SFTON3D P021
SMOVL C00538 BC00538 V=100.0  +MOVJ EC00538
SFTOF3D
MOVL C00539 BC00539 V=400.0  +MOVJ EC00539 VJ=100.00
SFTON3D P021
SMOVL C00540 BC00540 V=166.7 PL=0  +MOVJ EC00540
SREFP 1 C00541 BC00541  +REFP EC00541
SREFP 2 C00542 BC00542  +REFP EC00542
MACRO1 MJ#(0) ARGF9
ARCON
SMOVL C00543 BC00543 V=12.5  +MOVJ EC00543
SMOVL C00544 BC00544 V=12.5  +MOVJ EC00544
ARCOF
SFTOF3D
MOVL C00545 BC00545 V=400.0  +MOVJ EC00545 VJ=100.00
MOVL C00546 BC00546 V=1000.0  +MOVJ EC00546 VJ=100.00
MOVJ C00547 BC00547 VJ=100.00  +MOVJ EC00547 VJ=100.00
MOVJ C00548 BC00548 VJ=100.00  +MOVJ EC00548 VJ=100.00
MOVJ C00549 BC00549 VJ=100.00  +MOVJ EC00549 VJ=100.00
'2
'Path W3693
SFTOF3D
MOVJ C00550 BC00550 VJ=100.00  +MOVJ EC00550 VJ=100.00
MACRO1 MJ#(0) ARGF6
SFTON3D P060
SMOVL C00551 BC00551 V=166.7  +MOVJ EC00551
ARCON
SMOVL C00552 BC00552 V=8.3  +MOVJ EC00552
SMOVL C00553 BC00553 V=8.3  +MOVJ EC00553
SMOVL C00554 BC00554 V=8.3  +MOVJ EC00554
ARCOF
SMOVL C00555 BC00555 V=166.7  +MOVJ EC00555
SMOVL C00556 BC00556 V=333.3  +MOVJ EC00556
MACRO1 MJ#(0) ARGF14
SFTON3D P061
SMOVL C00557 BC00557 V=166.7  +MOVJ EC00557
ARCON
SMOVL C00558 BC00558 V=10.0  +MOVJ EC00558
ARCOF
SFTOF3D
SMOVL C00559 BC00559 V=416.7  +MOVJ EC00559
MOVJ C00560 BC00560 VJ=100.00  +MOVJ EC00560 VJ=25.00
MOVL C00561 BC00561 V=400.0  +MOVJ EC00561 VJ=100.00
SFTON3D P023
SMOVL C00562 BC00562 V=166.7 PL=0  +MOVJ EC00562
SREFP 1 C00563 BC00563  +REFP EC00563
SREFP 2 C00564 BC00564  +REFP EC00564
MACRO1 MJ#(0) ARGF9
ARCON
SMOVL C00565 BC00565 V=11.7  +MOVJ EC00565
ARCOF
SFTOF3D
MOVL C00566 BC00566 V=400.0  +MOVJ EC00566 VJ=100.00
MOVL C00567 BC00567 V=1000.0  +MOVJ EC00567 VJ=100.00
'Path W3694
SFTOF3D
MOVJ C00568 BC00568 VJ=20.00  +MOVJ EC00568 VJ=0.78
MOVJ C00569 BC00569 VJ=100.00  +MOVJ EC00569 VJ=100.00
MOVL C00570 BC00570 V=400.0  +MOVJ EC00570 VJ=100.00
SFTON3D P023
SMOVL C00571 BC00571 V=166.7 PL=0  +MOVJ EC00571
SREFP 1 C00572 BC00572  +REFP EC00572
SREFP 2 C00573 BC00573  +REFP EC00573
ARCON
SMOVL C00574 BC00574 V=11.7  +MOVJ EC00574
ARCOF
SFTOF3D
MOVL C00575 BC00575 V=400.0  +MOVJ EC00575 VJ=100.00
MOVL C00576 BC00576 V=1000.0  +MOVJ EC00576 VJ=100.00
MOVJ C00577 BC00577 VJ=100.00  +MOVJ EC00577 VJ=100.00
MOVJ C00578 BC00578 VJ=100.00  +MOVJ EC00578 VJ=100.00
MOVJ C00579 BC00579 VJ=100.00  +MOVJ EC00579 VJ=100.00
MOVJ C00580 BC00580 VJ=100.00  +MOVJ EC00580 VJ=100.00
SFTOF3D
MOVJ C00581 BC00581 VJ=100.00  +MOVJ EC00581 VJ=100.00
SFTOF3D
MOVJ C00582 BC00582 VJ=100.00  +MOVJ EC00582 VJ=100.00
MOVL C00583 BC00583 V=666.7  +MOVJ EC00583 VJ=100.00
SFTON3D P021
MACRO1 MJ#(0) ARGF9
SMOVL C00584 BC00584 V=166.7 PL=0  +MOVJ EC00584
SREFP 1 C00585 BC00585  +REFP EC00585
SREFP 2 C00586 BC00586  +REFP EC00586
ARCON
SMOVL C00587 BC00587 V=11.7  +MOVJ EC00587
ARCOF
SFTOF3D
MOVL C00588 BC00588 V=400.0  +MOVJ EC00588 VJ=100.00
MOVL C00589 BC00589 V=1000.0  +MOVJ EC00589 VJ=100.00
MOVJ C00590 BC00590 VJ=100.00  +MOVJ EC00590 VJ=100.00
MOVJ C00591 BC00591 VJ=100.00  +MOVJ EC00591 VJ=100.00
MOVJ C00592 BC00592 VJ=100.00  +MOVJ EC00592 VJ=100.00
MOVJ C00593 BC00593 VJ=100.00  +MOVJ EC00593 VJ=100.00
MOVJ C00594 BC00594 VJ=100.00  +MOVJ EC00594 VJ=100.00
'Path W3697
SFTOF3D
MOVJ C00595 BC00595 VJ=100.00  +MOVJ EC00595 VJ=100.00
MOVL C00596 BC00596 V=666.7  +MOVJ EC00596 VJ=100.00
SMOVL C00597 BC00597 V=133.3 PL=0  +MOVJ EC00597
SREFP 1 C00598 BC00598  +REFP EC00598
SREFP 2 C00599 BC00599  +REFP EC00599
ARCON
SMOVL C00600 BC00600 V=11.7  +MOVJ EC00600
ARCOF
MOVL C00601 BC00601 V=400.0  +MOVJ EC00601 VJ=100.00
MOVL C00602 BC00602 V=1000.0  +MOVJ EC00602 VJ=100.00
'Path W3698
SFTOF3D
MOVJ C00603 BC00603 VJ=100.00  +MOVJ EC00603 VJ=100.00
MOVL C00604 BC00604 V=400.0  +MOVJ EC00604 VJ=100.00
SFTON3D P023
SMOVL C00605 BC00605 V=133.3 PL=0  +MOVJ EC00605
SREFP 1 C00606 BC00606  +REFP EC00606
SREFP 2 C00607 BC00607  +REFP EC00607
ARCON
SMOVL C00608 BC00608 V=11.7  +MOVJ EC00608
ARCOF
SFTOF3D
MOVL C00609 BC00609 V=400.0  +MOVJ EC00609 VJ=100.00
MOVL C00610 BC00610 V=1000.0  +MOVJ EC00610 VJ=100.00
'5
MOVJ C00611 BC00611 VJ=100.00  +MOVJ EC00611 VJ=100.00
MOVJ C00612 BC00612 VJ=100.00  +MOVJ EC00612 VJ=100.00
MOVJ C00613 BC00613 VJ=100.00  +MOVJ EC00613 VJ=100.00
SFTOF3D
MOVJ C00614 BC00614 VJ=100.00  +MOVJ EC00614 VJ=100.00
MOVL C00615 BC00615 V=400.0  +MOVJ EC00615 VJ=100.00
SFTON3D P022
SMOVL C00616 BC00616 V=133.3 PL=0  +MOVJ EC00616
SREFP 1 C00617 BC00617  +REFP EC00617
SREFP 2 C00618 BC00618  +REFP EC00618
ARCON
SMOVL C00619 BC00619 V=11.7  +MOVJ EC00619
ARCOF
SFTOF3D
MOVL C00620 BC00620 V=400.0  +MOVJ EC00620 VJ=100.00
MOVL C00621 BC00621 V=1000.0  +MOVJ EC00621 VJ=100.00
'6
MOVJ C00622 BC00622 VJ=100.00  +MOVJ EC00622 VJ=100.00
MOVJ C00623 BC00623 VJ=100.00  +MOVJ EC00623 VJ=100.00
MOVJ C00624 BC00624 VJ=100.00  +MOVJ EC00624 VJ=100.00
'Path W3701
SFTOF3D
MOVJ C00625 BC00625 VJ=100.00  +MOVJ EC00625 VJ=100.00
MOVJ C00626 BC00626 VJ=100.00  +MOVJ EC00626 VJ=100.00
MOVL C00627 BC00627 V=400.0  +MOVJ EC00627 VJ=100.00
SFTON3D P023
SMOVL C00628 BC00628 V=166.7 PL=0  +MOVJ EC00628
SREFP 1 C00629 BC00629  +REFP EC00629
SREFP 2 C00630 BC00630  +REFP EC00630
ARCON
SMOVL C00631 BC00631 V=11.7  +MOVJ EC00631
ARCOF
SFTOF3D
MOVL C00632 BC00632 V=400.0  +MOVJ EC00632 VJ=100.00
MOVL C00633 BC00633 V=1000.0  +MOVJ EC00633 VJ=100.00
'Path W3702
SFTOF3D
MOVJ C00634 BC00634 VJ=100.00  +MOVJ EC00634 VJ=100.00
MOVL C00635 BC00635 V=400.0  +MOVJ EC00635 VJ=100.00
SFTON3D P023
SMOVL C00636 BC00636 V=166.7 PL=0  +MOVJ EC00636
SREFP 1 C00637 BC00637  +REFP EC00637
SREFP 2 C00638 BC00638  +REFP EC00638
ARCON
SMOVL C00639 BC00639 V=12.5  +MOVJ EC00639
ARCOF
SFTOF3D
MOVL C00640 BC00640 V=400.0  +MOVJ EC00640 VJ=100.00
MOVL C00641 BC00641 V=1000.0  +MOVJ EC00641 VJ=100.00
SFTOF3D
MOVJ C00642 BC00642 VJ=100.00  +MOVJ EC00642 VJ=100.00
MOVL C00643 BC00643 V=400.0  +MOVJ EC00643 VJ=100.00
MACRO1 MJ#(0) ARGF9
SFTON3D P022
SMOVL C00644 BC00644 V=166.7 PL=0  +MOVJ EC00644
SREFP 1 C00645 BC00645  +REFP EC00645
SREFP 2 C00646 BC00646  +REFP EC00646
ARCON
SMOVL C00647 BC00647 V=11.7  +MOVJ EC00647
ARCOF
SFTOF3D
MOVL C00648 BC00648 V=400.0  +MOVJ EC00648 VJ=100.00
MOVL C00649 BC00649 V=1000.0  +MOVJ EC00649 VJ=100.00
'8
'Path W3705
SFTOF3D
MOVJ C00650 BC00650 VJ=100.00  +MOVJ EC00650 VJ=100.00
MOVL C00651 BC00651 V=400.0  +MOVJ EC00651 VJ=100.00
SFTON3D P022
SMOVL C00652 BC00652 V=166.7 PL=0  +MOVJ EC00652
SREFP 1 C00653 BC00653  +REFP EC00653
SREFP 2 C00654 BC00654  +REFP EC00654
MACRO1 MJ#(0) ARGF14
ARCON
SMOVL C00655 BC00655 V=10.0  +MOVJ EC00655
ARCOF
SFTOF3D
MOVL C00656 BC00656 V=400.0  +MOVJ EC00656 VJ=100.00
MOVL C00657 BC00657 V=1000.0  +MOVJ EC00657 VJ=100.00
'Path W3706
SFTOF3D
MOVJ C00658 BC00658 VJ=100.00  +MOVJ EC00658 VJ=100.00
MOVL C00659 BC00659 V=400.0  +MOVJ EC00659 VJ=100.00
SFTON3D P022
SMOVL C00660 BC00660 V=166.7 PL=0  +MOVJ EC00660
SREFP 1 C00661 BC00661  +REFP EC00661
SREFP 2 C00662 BC00662  +REFP EC00662
MACRO1 MJ#(0) ARGF9
ARCON
SMOVL C00663 BC00663 V=10.8  +MOVJ EC00663
ARCOF
SFTOF3D
MOVL C00664 BC00664 V=400.0  +MOVJ EC00664 VJ=100.00
MOVL C00665 BC00665 V=1000.0  +MOVJ EC00665 VJ=100.00
END
